TYPE RecipeList_Struct :
STRUCT
	ToolId: LREAL;
	PosX: LREAL;
	PosY: LREAL;
	PosZ: LREAL;
	Tool1: LREAL;
	Tool2: LREAL;
	Tool3: LREAL;
	GlueTime: LREAL;
	Velo: LREAL;
	Reserve: ARRAY[10..20] OF LREAL;
END_STRUCT
END_TYPE

(* stored: Version 1.1.0.1, ProductVersion 3.1.0.12
   DUT RecipeList_Struct: Id {7bc47c37-58e8-4f7d-8f90-0ca275f5eb05} *)
